{attribute 'OPC.UA.DA.JobMethod' := 'JobMethode_HorizontalMove'}
FUNCTION_BLOCK SST_CB_AS_HorizontalMove
VAR
	AlwaysTrue : BOOL := TRUE;
	// Used for debugging purposes to display InputArguments of method call
	MethodCall_HorizontalMove : BOOL := FALSE; // used to store InputArg "MethodCall" from Start() method
	Direction : BOOL := FALSE;
//	TS_EndschalterEntlastung : BOOL;
	callCounterStart : ULINT; // counts how many times the Start() method has been called
	callCounterCheckState : ULINT; // counts how many times the CheckState() method has been called
	callCounterAbort : ULINT; // counts how many times the Abort() method has been called
	
	// Variables to determine if a job has been started (Start() method has been called) or finished
	jobRunning : BOOL;
	jobFinished : BOOL;

	// State machine variable
	state : UDINT;
	
	//Variablen des Transport FBs
	ResetCall : BOOL := FALSE;	
	JobMethode_Name : AxisControl_MultipleInputSensors;
END_VAR
	
VAR_INPUT
	NotAusSignal: BOOL;
	LightSensor_01 : BOOL;
	LightSensor_02 : BOOL;
	TS_Endschalter_01 : BOOL;
	TS_Endschalter_02 : BOOL;
	TOF_Time_Motoransteuerung : TIME;
	TOF_Time_EndschalterEntlastung : TIME;
END_VAR

VAR_OUTPUT
	Motor_Ansteuerung01 : BOOL;
	Motor_Ansteuerung02 : BOOL;
END_VAR

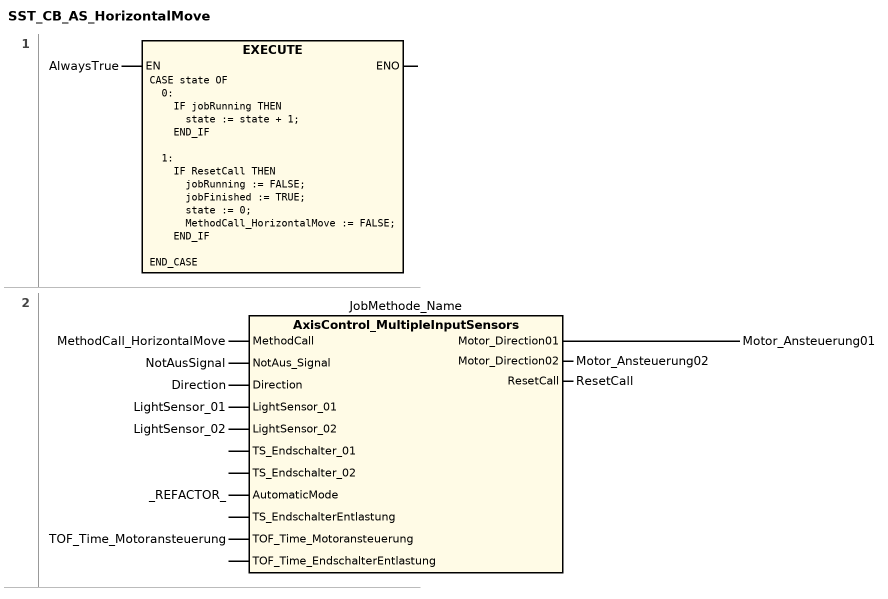
// NETWORK 1
IF AlwaysTrue THEN
    CASE state OF
    	0:
    		IF jobRunning THEN
    			state := state + 1;
    		END_IF
    		
    	1:
    		IF ResetCall THEN
    			jobRunning := FALSE;
    			jobFinished := TRUE;
    			state := 0;
    			MethodCall_HorizontalMove := FALSE;
    		END_IF
    		
    END_CASE
END_IF

// NETWORK 2
JobMethode_Name(
    MethodCall := MethodCall_HorizontalMove,
    NotAus_Signal := NotAusSignal,
    Direction := Direction,
    LightSensor_01 := LightSensor_01,
    LightSensor_02 := LightSensor_02,
    AutomaticMode := _REFACTOR_,
    TOF_Time_Motoransteuerung := TOF_Time_Motoransteuerung,
    Motor_Direction02 => Motor_Ansteuerung02,
    ResetCall => ResetCall); // AxisControl_MultipleInputSensors
Motor_Ansteuerung01 := JobMethode_Name.Motor_Direction01;

{attribute 'TcRpcEnable' := '1'}
METHOD Abort : HRESULT
VAR_INPUT
	hdl : UDINT; // Do not change, used by server.
END_VAR
callCounterAbort := callCounterAbort + 1;
END_METHOD

{attribute 'TcRpcEnable' := '1'}
METHOD CheckState : HRESULT
VAR_INPUT
	hdl : UDINT; // Do not change, used by server.
END_VAR
VAR_OUTPUT
	bBusy : BOOL; // Do not change. Used by server to find out if the job is finished
	
	// List of OutputArguments for OPC UA method, may be customized
	State : BOOL; // Abgeschlossener MethodCall
	MethodCall: BOOL; //Input Recall
END_VAR
callCounterCheckState := callCounterCheckState + 1;
IF NOT jobFinished THEN
	bBusy := TRUE; // job is not finished yet
	CheckState := 0; // no error
ELSE
	bBusy := FALSE; // job is finished
	CheckState := 0; // done, no error occured during execution (OPC UA StatusCode "GOOD")
	jobFinished := FALSE;
	State := ResetCall;
	MethodCall := MethodCall_HorizontalMove;
END_IF
END_METHOD

{attribute 'TcRpcEnable' := '1'}
METHOD Start : HRESULT
VAR_INPUT
	// List of InputArguments for OPC UA method, may be customized
	MethodCall : BOOL; // some description
	DirectionPoint : BOOL;
//	EndschalterEntlastung : BOOL;	
END_VAR
VAR_OUTPUT
	hdl : UDINT; // Do not change, used by server.
END_VAR
callCounterStart := callCounterStart + 1;

MethodCall_HorizontalMove := MethodCall;
DirectionPoint := Direction;
//EndschalterEntlastung := EndschalterEntlastung;

jobRunning := TRUE;
Start := 0; // no error occured, e.g. while parsing the input arguments (0 = OPC UA StatusCode "GOOD")
END_METHOD

END_FUNCTION_BLOCK

(* stored: Version 1.1.0.1, ProductVersion 3.1.4024.15
   POU SST_CB_AS_HorizontalMove: Id {e20621e3-ba6b-4a13-819b-927624ce5ea9}, SpecialFunc None
   Method Abort: Id {5f94a12f-2a1f-4f42-a4e3-7ba9fb1ec2c7}
   Method CheckState: Id {997d9f38-b8aa-42e5-ae89-b3836326f5e7}
   Method Start: Id {2175a7f6-5ad3-499e-b970-80733b0797e4} *)
